(*******************************************************************************
                          protoc-gen-twincat V0.0.0.0                           
                  https://github.com/TcHaxx/protoc-gen-twincat                  
*******************************************************************************)
TYPE ST_Baz :
STRUCT
	value : UDINT;
	name : STRING;
END_STRUCT
END_TYPE

(* stored: Version 1.1.0.1
   DUT ST_Baz: Id {dc237215-8bf7-44a9-ae70-fd15e9b3ce81} *)
